{attribute 'qualified_only'}
{attribute 'strict'}
{attribute 'to_string'}
TYPE DUT_Command_VisionType :
(
	Calibrate := 0,
    Acquire := 1,
    LocatePart :=2
);
END_TYPE

(* stored: Version 1.1.0.1
   EnumerationTextList DUT_Command_VisionType: Id {05d30690-68b6-445a-a0fb-0f99b45b92a3} *)
